(* CoDeSys 2.3 export: PWMTIMER.EXP *)

(* POU Components/OnOff/PWMTimer, ST *)
FUNCTION_BLOCK PWMTimer
VAR_INPUT
	start:BOOL;
	onTimeSetup:INT;
	offTimeSetup:INT;
END_VAR
VAR_OUTPUT
	output:BOOL;
END_VAR
VAR
	onTimer:Delay;
	offTimer:Delay;
END_VAR
onTimer.timeSetup:=onTimeSetup;
offTimer.timeSetup:=offTimeSetup;

onTimer(start:=start);
offTimer(start:=onTimer.afterTime);
onTimer.resetTime:=offTimer.afterTimeImpulse;
output:= onTimer.untilTimePass;
END_FUNCTION_BLOCK
